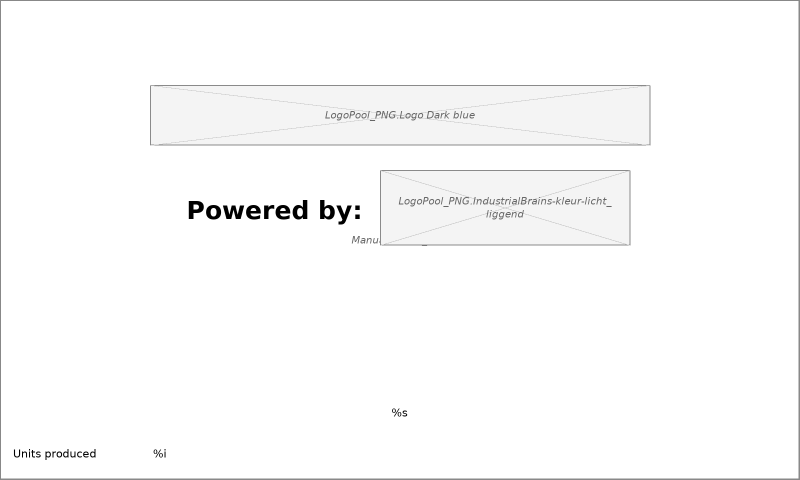
VISUALIZATION LogoScreenBliss_PNG  // 800x480
VAR_INPUT
	nUnitsProduced	: UDINT; // HMI Main total units produced
END_VAR
VAR_IN_OUT
	bCmdManual		: BOOL ; // HMI switch to manual mode
END_VAR
    Frame (0,0 800x480)
        shows ManualButton_PNG(bCmdManual := bCmdManual)
    Image (150,85 500x60), image: LogoPool_PNG.Logo Dark blue
    Image (380,170 250x75), image: LogoPool_PNG.IndustrialBrains-kleur-licht_liggend
    Textfield (183,404 433x18), "%s", tooltip "Operator messagages", text variable: GVL_Message.sOPeratorMessage
    Textfield (110,439 100x30), "%i", text variable: nUnitsProduced
    Label (10,439 100x30), "Units produced"
    Label (179,150 200x120), "Powered by:"
END_VISUALIZATION

(* stored: Version 1.1.0.1, ProductVersion 3.1.4024.11
   Visu LogoScreenBliss_PNG: Id {b7a98265-18b5-4c84-9f59-a6c5d1c46c59} *)
